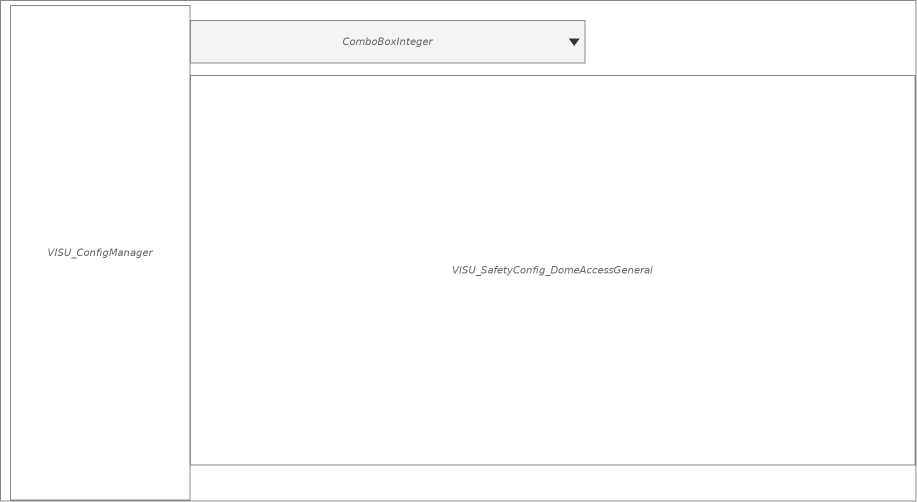
VISUALIZATION VISU_SafetyConfig  // 917x502
VAR_IN_OUT
    editable : SafetyConfig;
	active : SafetyConfig;
    mgr : ConfigManager;
    mgrWidget : ConfigManagerWidget;
    widget : SafetyWidget;
END_VAR
    Frame (10,5 180x495)
        shows VISU_ConfigManager(mgr := mgr, widget := mgrWidget)
    ComboBoxInteger (190,20 395x43), variable: widget.activeConfigTab, text list: 'SafetyConfigTabsTextList'
    Frame (190,75 725x390), frame switch variable: widget.activeConfigTab
        shows VISU_SafetyConfig_DomeAccessGeneral(editable := editable.domeAccess, active := active.domeAccess)
        shows VISU_SafetyConfig_DomeAccessAlert(editable := editable.domeAccess.bypassingSound, active := active.domeAccess.bypassingSound)
        shows VISU_SafetyConfig_DomeAccessAlert(editable := editable.domeAccess.bypassedPermanentlyVisual, active := active.domeAccess.bypassedPermanentlyVisual)
        shows VISU_SafetyConfig_DomeAccessAlert(editable := editable.domeAccess.doorsOpenedWhenEnteringSound, active := active.domeAccess.doorsOpenedWhenEnteringSound)
        shows VISU_SafetyConfig_DomeAccessAlert(editable := editable.domeAccess.doorsOpenedWhenLeavingSound, active := active.domeAccess.doorsOpenedWhenLeavingSound)
        shows VISU_SafetyConfig_DomeAccessAlert(editable := editable.domeAccess.leavingWhenDoorsClosedSound, active := active.domeAccess.leavingWhenDoorsClosedSound)
        shows VISU_SafetyConfig_DomeAccessAlert(editable := editable.domeAccess.leavingWhenDoosOpenedSound, active := active.domeAccess.leavingWhenDoosOpenedSound)
        shows VISU_SafetyConfig_DomeAccessAlert(editable := editable.domeAccess.doorsOpenedVisual, active := active.domeAccess.doorsOpenedVisual)
        shows VISU_M1Config_Axial_AverageForce(editable := editableConfig.axialSupport, active := activeConfig.axialSupport)
        shows VISU_MeasurementConfig(active := activeConfig.inclinometerVoltage, editable := editableConfig.inclinometerVoltage)
        p2735656198: currentFocalStationPosition
END_VISUALIZATION

(* stored: Version 1.1.0.1, ProductVersion 3.1.4019.2
   Visu VISU_SafetyConfig: Id {9ff18b2b-40b1-4ae2-b2e7-ab6889af6511} *)
